FUNCTION_BLOCK APPEND_STRING_2 (* Service Interface Function Block Type *)
  (* Standard: 61499-2 *)
  (* Version 0.0, 2012-06-20, 4DIAC-IDE, 4DIAC-Consortium *)
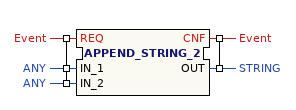
  EVENT_INPUT
    REQ WITH IN_1, IN_2; (* Service Request *)
  END_EVENT
  EVENT_OUTPUT
    CNF WITH OUT; (* Confirmation of Requested Service *)
  END_EVENT
  VAR_INPUT
    IN_1 : ANY; (* Data Input 1 (value is converted to String) *)
    IN_2 : ANY; (* Data Input 2 (value is converted to String) *)
  END_VAR
  VAR_OUTPUT
    OUT : STRING; (* Concatenated output string *)
  END_VAR
  (* Service APPLICATION/RESOURCE: Service Interface Function Block Type *)
END_FUNCTION_BLOCK
